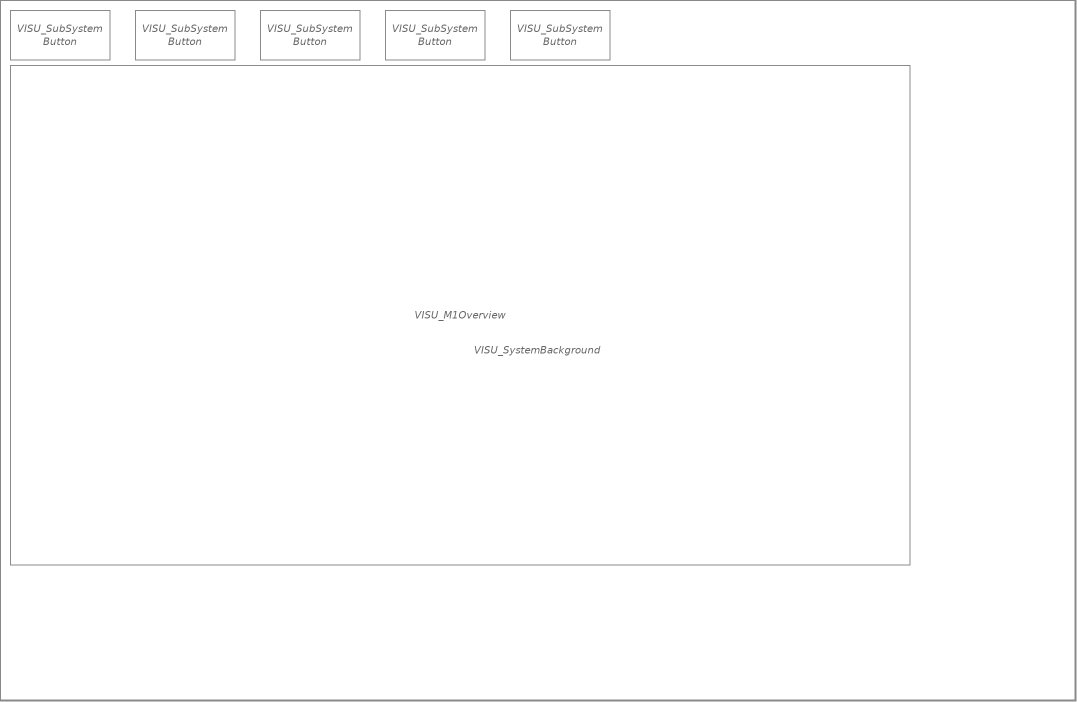
VISUALIZATION VISU_M1  // 1077x702
VAR_IN_OUT
	ref : M1;
    widget : M1Widget;
END_VAR
    Frame (0,0 1075x700)
        shows VISU_SystemBackground(color := widget.actualStatus.color)
    Frame (10,65 900x500)
        shows VISU_M1Overview(ref := ref, widget := widget)
        shows VISU_M1RadialSupport(ref := ref.parts.radialSupport, widget := widget.radialSupport, m1Ref := ref, m1Widget := widget)
        shows VISU_M1AxialSupport(ref := ref.parts.axialSupport, widget := widget.axialSupport, m1Ref := ref, m1Widget := widget)
        shows VISU_M1M2IO(ref := ref.parts.io, widget := widget.io)
        shows VISU_M1Config(editableConfig := ref.editableConfig, activeConfig := ref.config, mgr := ref.parts.configManager, mgrWidget := widget.configManager, activeTab := widget.activeConfigTab)
        p701045219: ref.editableConfig
        p2690442461: ref.config
        p942769723: ref.parts.configManager
        p2963374678: widget.configManager
        p459268616: widget
    Frame (10,10 100x50)
        shows VISU_SubSystemButton(widget := widget.button_overview)
        OnMouseClick: FrameSelectionChange Selection=SelectedFrame=b1e9e4b0-bf3d-440f-90c5-cb513105ccf1, GlobSel=AssignType=Directly, SelType=Locally
        OnMouseClick: execute { widget.activeTab := M1Tabs.OVERVIEW; }
    Frame (135,10 100x50)
        shows VISU_SubSystemButton(widget := widget.button_radial)
        OnMouseClick: FrameSelectionChange Selection=SelectedFrame=b1e9e4b0-bf3d-440f-90c5-cb513105ccf1, Selection=1, GlobSel=AssignType=Directly, SelType=Locally
        OnMouseClick: execute { widget.activeTab := M1Tabs.RADIAL; }
    Frame (260,10 100x50)
        shows VISU_SubSystemButton(widget := widget.button_axial)
        OnMouseClick: FrameSelectionChange Selection=SelectedFrame=b1e9e4b0-bf3d-440f-90c5-cb513105ccf1, Selection=2, GlobSel=AssignType=Directly, SelType=Locally
        OnMouseClick: execute { widget.activeTab := M1Tabs.AXIAL; }
    Frame (385,10 100x50)
        shows VISU_SubSystemButton(widget := widget.button_io)
        OnMouseClick: FrameSelectionChange Selection=SelectedFrame=b1e9e4b0-bf3d-440f-90c5-cb513105ccf1, Selection=3, GlobSel=AssignType=Directly, SelType=Locally
        OnMouseClick: execute { widget.activeTab := M1Tabs.IO; }
    Frame (510,10 100x50)
        shows VISU_SubSystemButton(widget := widget.button_config)
        OnMouseClick: FrameSelectionChange Selection=SelectedFrame=b1e9e4b0-bf3d-440f-90c5-cb513105ccf1, Selection=4, GlobSel=AssignType=Directly, SelType=Locally
        OnMouseClick: execute { widget.activeTab := M1Tabs.CONFIG; }
END_VISUALIZATION

(* stored: Version 1.1.0.1, ProductVersion 3.1.4019.2
   Visu VISU_M1: Id {8ee338af-6eaf-4829-b2a3-c7c87458c2ed} *)
